% RSLogix 500 project 7.5.RSS, saved by version 8.30.00.16 %
PROJECT "7.5"    % processor: Bul.1763 MicroLogix 1100 Series B %

PROGRAM FILES
  LAD 2   5 rungs

DATA FILES
  O0 OUTPUT  4 elements
  I1 INPUT  6 elements
  S2 STATUS  66 elements
  B3 BINARY  1 elements
  T4 TIMER  2 elements
  C5 COUNTER  1 elements
  R6 CONTROL  1 elements
  N7 INTEGER  1 elements
  F8 FLOAT  1 elements

LADDER 2
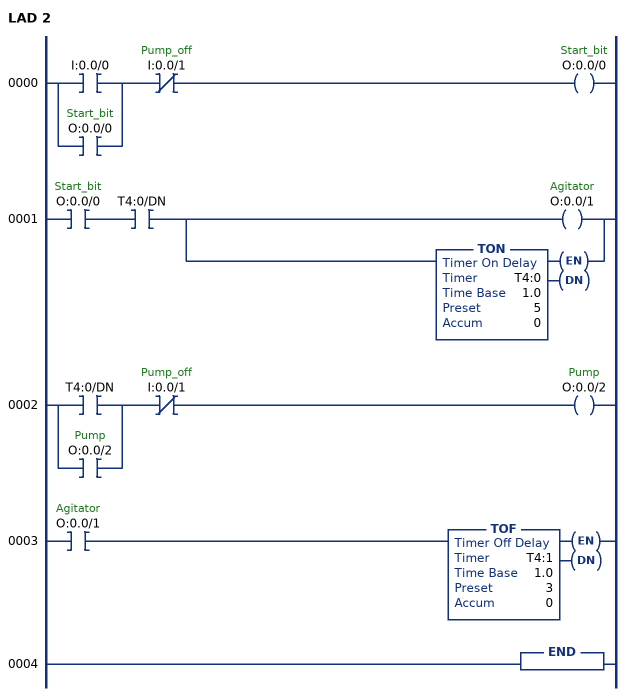
% Rung: 0 %
SOR BST XIC I:0.0/0 NXB XIC O:0.0/0 BND XIO I:0.0/1 OTE O:0.0/0 EOR
%   O:0.0/0  "Start_bit" %
%   I:0.0/1  "Pump_off" %
% Rung: 1 %  % edit flag set %
SOR XIC O:0.0/0 XIC T4:0/DN BST OTE O:0.0/1 NXB TON T4:0 1.0 5 0 BND EOR
%   O:0.0/0  "Start_bit" %
%   O:0.0/1  "Agitator" %
% Rung: 2 %
SOR BST XIC T4:0/DN NXB XIC O:0.0/2 BND XIO I:0.0/1 OTE O:0.0/2 EOR
%   O:0.0/2  "Pump" %
%   I:0.0/1  "Pump_off" %
% Rung: 3 %
SOR XIC O:0.0/1 TOF T4:1 1.0 3 0 EOR
%   O:0.0/1  "Agitator" %
% Rung: 4 %
SOR END EOR

DATA TABLE (non-zero values as saved)
DATA T4
% .PRE .ACC %
% T4:0 % 5 0
% T4:1 % 3 0
